TYPE ST_HmiStatistics :
STRUCT
    udiTotalCycles          : UDINT;
    udiTotalPass            : UDINT;
    udiTotalFail            : UDINT;
    udiEquipmentFaults      : UDINT;
    udiIndexFaults          : UDINT;
    udiSafetyStops          : UDINT;
    udiAbortedCycles        : UDINT;
    dtLastCycleCompleted    : DATE_AND_TIME;
END_STRUCT
END_TYPE

(* stored: Version 1.1.0.1, ProductVersion 3.1.4026.18
   DUT ST_HmiStatistics: Id {ca8058d7-b002-43e2-934b-a3a4b1017cc2} *)
